FUNCTION fSetPar : LREAL
VAR_INPUT
	///factor * SetValue
	In_dinSetValue: DINT;
	/// % from SetValue
	In_dinSetValue_per: DINT;
END_VAR
VAR
	/// every value is scaled with 10
	dinFactor: DINT := 10;
END_VAR

fSetPar := DINT_TO_LREAL((In_dinSetValue*In_dinSetValue_per) /(10*100));

END_FUNCTION

(* stored: Version 1.1.0.1, ProductVersion 3.1.0.25
   POU fSetPar_1: Id {d4385cb6-bc46-43d2-92e0-b36be35e0f68} *)
